{attribute 'qualified_only'}
{attribute 'strict'}
TYPE SynchronizationType :
(
  Phase, // Phase synchronize the DoFs when possible, else fallback to "Time" strategy
  TimeSync, // Always synchronize the DoFs to reach the target at the same time (Default)
  TimeIfNecessarySync, // Synchronize only when necessary (e.g. for non-zero target velocity or acceleration)
  None // Calculate every DoF independently
);
END_TYPE

(* stored: Version 1.1.0.1
   DUT SynchronizationType: Id {c2f32290-f62f-4354-9b4e-71d37ff75e54} *)
